Staubli VAL3: reset.pgx

public program reset()
begin
  // This program resets the conveyor libraries. This reset consist of :
  // - flushing the conveyor's queue
  //
  // Created 29-05-08                                  C.CURRIVAND
  //----------------------------------------------------------------
  bResetConv=true
  call enc:reset()
end
